PROGRAM GEMMA
VAR
	STEP_A6: INT := 0;
	DELAY_EJECTION_CARRIERS: TON;
	EJECT_CARRIERS: BOOL;
	F2_END: BOOL;
	STEP: STRING(20);
END_VAR

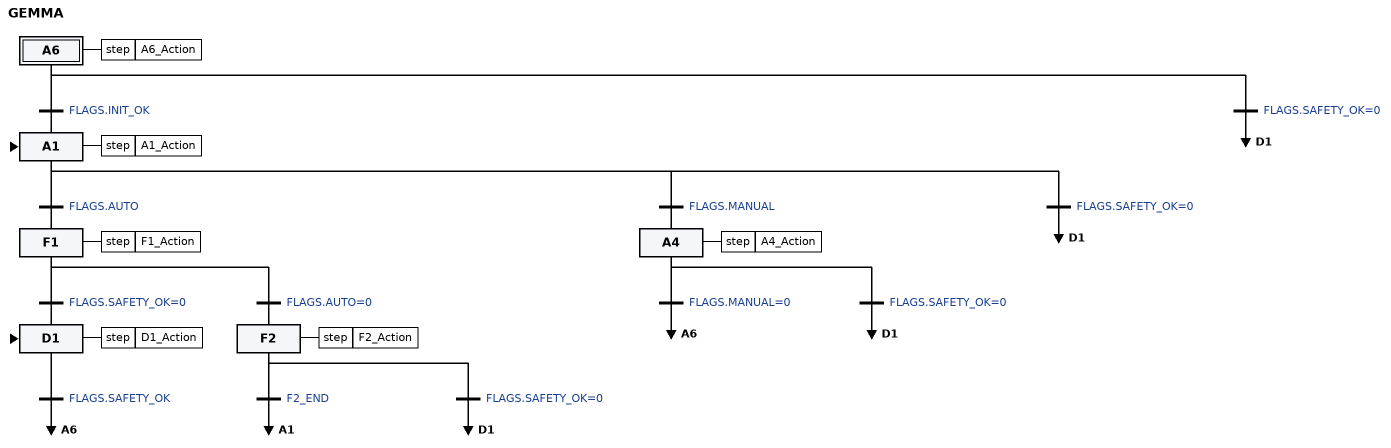
INITIAL_STEP A6_:  // name as stored: A6 
    A6_Action(N);  // step action
END_STEP
TRANSITION FROM A6_ TO A1
    := FLAGS.INIT_OK;
END_TRANSITION
TRANSITION FROM A6_ TO D1
    := FLAGS.SAFETY_OK=0;
END_TRANSITION
STEP A1:
    A1_Action(N);  // step action
END_STEP
TRANSITION FROM A1 TO F1
    := FLAGS.AUTO;
END_TRANSITION
TRANSITION FROM A1 TO A4
    := FLAGS.MANUAL;
END_TRANSITION
STEP A4:
    A4_Action(N);  // step action
END_STEP
TRANSITION FROM A4 TO A6
    := FLAGS.MANUAL=0;
END_TRANSITION
TRANSITION FROM A4 TO D1
    := FLAGS.SAFETY_OK=0;
END_TRANSITION
TRANSITION FROM A1 TO D1
    := FLAGS.SAFETY_OK=0;
END_TRANSITION
STEP F1:
    F1_Action(N);  // step action
END_STEP
TRANSITION FROM F1 TO D1
    := FLAGS.SAFETY_OK=0;
END_TRANSITION
TRANSITION FROM F1 TO F2
    := FLAGS.AUTO=0;
END_TRANSITION
STEP F2:
    F2_Action(N);  // step action
END_STEP
TRANSITION FROM F2 TO A1
    := F2_END;
END_TRANSITION
TRANSITION FROM F2 TO D1
    := FLAGS.SAFETY_OK=0;
END_TRANSITION
STEP D1:
    D1_Action(N);  // step action
END_STEP
TRANSITION FROM D1 TO A6
    := FLAGS.SAFETY_OK;
END_TRANSITION

ACTION A6_Action:
(**************************************************************
*
*
* Initialisation
*
*
***************************************************************)
STEP:='A6';

PMAX();
VAC();
Q1();
Q2();
(*CONVEYOR();*)


CASE STEP_A6 OF

0: (*Init*)
	STEP_A6:=STEP_A6+1;

1: (*Initialise valves and variables*)

	FLAGS.INIT_OK:=FALSE;
	FLAGS.INIT_CHECK_VALVES_SENSORS:=TRUE;

	FLAGS.VAC_RELEASE_CARRIER:=FALSE;
	FLAGS.Q1_RELEASE_CARRIER:=FALSE;
	FLAGS.Q2_RELEASE_CARRIER:=FALSE;
	FLAGS.PMAX_RELEASE_CARRIER:=FALSE;
	FLAGS.PRINT_RELEASE_CARRIER:=FALSE;

	FLAGS.MOTOR_Q1_INIT_OK:=FALSE;
	FLAGS.MOTOR_Q1_POSITION:=MOTOR_Q1_INITIAL_POS;

	VAC_DO.AIR_VALVE := FALSE;

	VAC_DO.ELECTR_CYLINDER := FALSE;
	VAC_DO.HYDRO_CYLINDER_BOT := FALSE;
	VAC_DO.HYDRO_CYLINDER_TOP := FALSE;

	VAC_DO.WAGON_LOCK_CYLINDER := FALSE;
	VAC_DO.WAGON_STOP_CYLINDER := FALSE;
	VAC_DO.WAGON_WAIT_CYLINDER := FALSE;

	VAC_DO.FLOW_STOP_VALVE := FALSE;
	VAC_DO.WATER_TANK_VALVE := FALSE;
	VAC_DO.PUMP_POWER := FALSE;
	VAC_DO.VACUUM_VALVE := FALSE;
	VAC_DO.WAGON_OPERATOR1:=TRUE;
	VAC_DO.WAGON_OPERATOR2:=TRUE;


	Q1_DO.ELECTR_CYLINDER := FALSE;
	Q1_DO.HYDRO_CYLINDER_BOT := FALSE;
	Q1_DO.HYDRO_CYLINDER_TOP := FALSE;
	Q1_DO.WAGON_LOCK_CYLINDER := FALSE;
	Q1_DO.WAGON_STOP_CYLINDER := FALSE;
	Q1_DO.WAGON_WAIT_CYLINDER := FALSE;
	Q1_DO.PUMP_POWER:=FALSE;
	Q1_DO.FLOW_STOP_BOTT:=FALSE;

	Q2_DO.ELECTR_CYLINDER := FALSE;
	Q2_DO.HYDRO_CYLINDER_BOT := FALSE;
	Q2_DO.HYDRO_CYLINDER_TOP := FALSE;
	Q2_DO.WAGON_LOCK_CYLINDER := FALSE;
	Q2_DO.WAGON_STOP_CYLINDER := FALSE;
	Q2_DO.WAGON_WAIT_CYLINDER := FALSE;
	Q2_DO.PUMP_POWER:=FALSE;
	Q2_DO.FLOW_STOP_BOTT:=TRUE;

	PMAX_DO.ELECTR_CYLINDER := FALSE;
	PMAX_DO.HYDRO_CYLINDER_BOT := FALSE;
	PMAX_DO.HYDRO_CYLINDER_TOP := FALSE;
	PMAX_DO.WAGON_LOCK_CYLINDER := FALSE;
	PMAX_DO.WAGON_STOP_CYLINDER := FALSE;
	PMAX_DO.WAGON_WAIT_CYLINDER := FALSE;
	PMAX_DO.PUMP_POWER:=FALSE;
	PMAX_DO.FLOW_STOP_BOTT:=FALSE;

	PRINT_DO.WAGON_LOCK_CYLINDER := FALSE;
	PRINT_DO.WAGON_STOP_CYLINDER := FALSE;
	PRINT_DO.WAGON_WAIT_CYLINDER := FALSE;


	STEP_A6:=STEP_A6+1;

2: (*Start AIR and wait for ejection of all carriers on the conveyor*)

	VAC_DO.AIR_VALVE := TRUE;
	POW_DO.CONVEYOR_RELAIS := TRUE;
	EJECT_CARRIERS:=TRUE;

	STEP_A6:=STEP_A6+1;

3: (* Wait carriers ejection *)

	IF DELAY_EJECTION_CARRIERS.Q THEN
		EJECT_CARRIERS:=FALSE;
		STEP_A6:=STEP_A6+1;
	END_IF;

4:(*Check valves sensors A IMPLEMENTER PLUS TARD *)
	IF FLAGS.INIT_CHECK_VALVES_SENSORS THEN
		;(*CHECK_VALVES_SENSORS();*)
		STEP_A6:=STEP_A6+1;
	ELSE
		STEP_A6:=STEP_A6+1;
	END_IF;

5: (*End of init *)

	FLAGS.INIT_OK:=TRUE;


ELSE
    ;
END_CASE;

(* FBs *)
DELAY_EJECTION_CARRIERS(IN:=EJECT_CARRIERS , PT:= DELAY_EJECT_CARRIERS);
END_ACTION

ACTION F2_Action:
STEP := 'F2';

VAC();
CONVEYOR();

IF VAC.STEP=10 THEN

F2_END:=TRUE;

END_IF;
END_ACTION

ACTION A1_Action:
(***************************************************************************
*
* A1
*
****************************************************************************)
STEP := 'A1';

F2_END:=FALSE;
END_ACTION

ACTION F1_Action:
(*********************************************************
*
* F1
*
************************************************************)

STEP := 'F1';

(* Station VAC *)
IF PUMP_PARAMS.VAC_ENABLE THEN
	VAC();
ELSE
	FLAGS.VAC_RELEASE_CARRIER:=TRUE;
END_IF;

(* Station Q1 *)
IF PUMP_PARAMS.Q1_ENABLE THEN
	Q1();
ELSE
	FLAGS.Q1_RELEASE_CARRIER:=TRUE;
END_IF;

(* Station Q2 *)
IF PUMP_PARAMS.Q2_ENABLE THEN
	Q2();
ELSE
	FLAGS.Q2_RELEASE_CARRIER:=TRUE;
END_IF;

(* Station PMAX *)
IF PUMP_PARAMS.PMAX_ENABLE THEN
	PMAX();
ELSE
	FLAGS.PMAX_RELEASE_CARRIER:=TRUE;
END_IF;

(* Station PRINT *)
IF PUMP_PARAMS.PRINT_ENABLE THEN
	PRINT();
ELSE
	FLAGS.PRINT_RELEASE_CARRIER:=TRUE;
END_IF;



CONVEYOR();
END_ACTION

ACTION A4_Action:
STEP:= 'A4';
END_ACTION

ACTION D1_Action:
(*****************************************************************
*
* NOT AUS state
*
******************************************************************)

	STEP := 'D1';

	FLAGS.INIT_OK:=FALSE;
	FLAGS.MOTOR_Q1_INIT_OK:=FALSE;
	FLAGS.AUTO:=FALSE;
	FLAGS.MANUAL:=FALSE;


	VAC_DO.AIR_VALVE := FALSE;
	POW_DO.CONVEYOR_RELAIS:=FALSE;

	VAC_DO.ELECTR_CYLINDER := FALSE;
	VAC_DO.HYDRO_CYLINDER_BOT := FALSE;
	VAC_DO.HYDRO_CYLINDER_TOP := FALSE;
	VAC_DO.WAGON_LOCK_CYLINDER := FALSE;
	VAC_DO.WAGON_STOP_CYLINDER := FALSE;
	VAC_DO.WAGON_WAIT_CYLINDER := FALSE;
	VAC_DO.PUMP_POWER:=FALSE;
	VAC_DO.WAGON_OPERATOR1:=TRUE;
	VAC_DO.WAGON_OPERATOR2:=FALSE;

	Q1_DO.ELECTR_CYLINDER := FALSE;
	Q1_DO.HYDRO_CYLINDER_BOT := FALSE;
	Q1_DO.HYDRO_CYLINDER_TOP := FALSE;
	Q1_DO.WAGON_LOCK_CYLINDER := FALSE;
	Q1_DO.WAGON_STOP_CYLINDER := FALSE;
	Q1_DO.WAGON_WAIT_CYLINDER := FALSE;
	Q1_DO.PUMP_POWER:=FALSE;

	Q2_DO.ELECTR_CYLINDER := FALSE;
	Q2_DO.HYDRO_CYLINDER_BOT := FALSE;
	Q2_DO.HYDRO_CYLINDER_TOP := FALSE;
	Q2_DO.WAGON_LOCK_CYLINDER := FALSE;
	Q2_DO.WAGON_STOP_CYLINDER := FALSE;
	Q2_DO.WAGON_WAIT_CYLINDER := FALSE;
	Q2_DO.PUMP_POWER:=FALSE;

	PMAX_DO.ELECTR_CYLINDER := FALSE;
	PMAX_DO.HYDRO_CYLINDER_BOT := FALSE;
	PMAX_DO.HYDRO_CYLINDER_TOP := FALSE;
	PMAX_DO.WAGON_LOCK_CYLINDER := FALSE;
	PMAX_DO.WAGON_STOP_CYLINDER := FALSE;
	PMAX_DO.WAGON_WAIT_CYLINDER := FALSE;
	PMAX_DO.PUMP_POWER:=FALSE;


	PRINT_DO.WAGON_LOCK_CYLINDER	:= FALSE;
	PRINT_DO.WAGON_STOP_CYLINDER 	:= FALSE;
	PRINT_DO.WAGON_WAIT_CYLINDER	:= FALSE;
	PRINT_DO.EJECTION_CYLINDER_X	:=FALSE;
	PRINT_DO.EJECTION_CYLINDER_Z	:=FALSE;
	PRINT_DO.EJECTION_GRIPPER		:=FALSE;

	STEP_A6:=0;


	CONVEYOR();
END_ACTION

END_PROGRAM

(* stored: Version 1.1.0.1, ProductVersion 3.1.0.26
   POU GEMMA: Id {bac9d8d4-08ae-4540-8443-cc3993dc2ed6}
   Action A6_Action: Id {8ee0afff-21cf-4558-acc5-8748dee5e10c}
   Action F2_Action: Id {9fe8c460-0276-45ed-bfa2-51d01d80f836}
   Action A1_Action: Id {b3b9f24f-0656-42fe-9aad-87fba863aef2}
   Action F1_Action: Id {bb59ae76-f3f1-49bf-a11f-fceddee3723a}
   Action A4_Action: Id {dac6ddbc-a835-43c8-8757-2e67ae276be1}
   Action D1_Action: Id {e7b47e9e-9f98-463e-b838-606d9c8666e7} *)
